// Mitsubishi GX Works2 project: 20150611   PLC: Q03UDV

PROGRAM P1
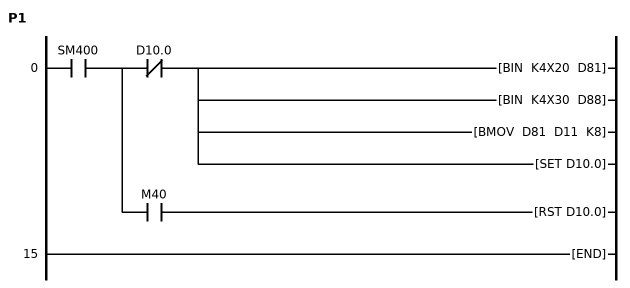
0     LD      SM400
      MPS
      ANI     D10.0
      BIN     K4X20 D81
      BIN     K4X30 D88
      BMOV    D81 D11 K8
      SET     D10.0
      MPP
      AND     M40
      RST     D10.0
15    END
END_PROGRAM

PROGRAM P2
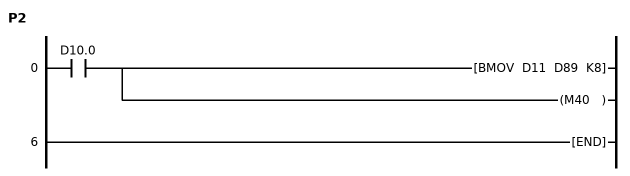
0     LD      D10.0
      BMOV    D11 D89 K8
      OUT     M40
6     END
END_PROGRAM
